TYPE EtcSlaveBase_82538BE2 :
STRUCT
END_STRUCT
END_TYPE

(* stored: Version 1.2.0.0, ProductVersion 3.1.4024.11
   DUT EtcSlaveBase_82538BE2: Id {91551ed6-a06f-4999-abdb-56ba097e5aeb} *)
